PROGRAM MAIN
VAR
	isFirstStart : BOOL := TRUE;
	valve_01 : FB_Valve_monostable;
	valve_02 : FB_Valve_monostable;
	
END_VAR

// Set IN(IT)
valve_01.MaxOpenCloseDuration := 180;// this setting can be reduced during test without the fysical Valve
valve_02.MaxOpenCloseDuration := 10;
GVL_VCM.valve01.TagName := 'Valve-01';
GVL_VCM.valve02.TagName := 'Valve-02';

IF isFirstStart THEN
	// Init the Valve at startup (for test/demo)
	GVL_VCM.ioValve01.I_isClosed := TRUE;
	GVL_VCM.ioValve02.I_isClosed := TRUE;
END_IF

// Do stuff
//create valve-01
valve_01(Valve:= GVL_VCM.valve01, I_O:= GVL_VCM.ioValve01);
//create valve-02
valve_02(Valve:= GVL_VCM.valve02, I_O:= GVL_VCM.ioValve02);

isFirstStart := FALSE;

END_PROGRAM

(* stored: Version 1.1.0.1, ProductVersion 3.1.4024.12
   POU MAIN: Id {b05310ae-f2a0-489f-aa66-207cf49f8ef4}, SpecialFunc None *)
